FUNCTION_BLOCK fbInverterPosCtrl
VAR_INPUT
	bHomingRdy		:	BOOL;
	bPosStart		:	BOOL;
	dTargetPosNum	:	DINT;
	i1stRPMfix		:	INT;
	i2ndRPMfix		:	INT;
	i2ndSpdRangefix	:	INT;
	iOffSetRangeFix	:	INT;
	iRatioFix			:	REAL;
	lrActualPosition	:	LREAL;

	iPos1			:	INT;
	iPos2			:	INT;
	iPos3			:	INT;
	iPos4			:	INT;
	iPos5			:	INT;
	iPos6			:	INT;
	iPos7			:	INT;
	iPos8			:	INT;
	iPos9			:	INT;
	iPos10			:	INT;
	iPos11			:	INT;
	iPos12			:	INT;
	iPos13			:	INT;
	iPos14			:	INT;
	iPos15			:	INT;
	iPos16			:	INT;
	iPos17			:	INT;
	iPos18			:	INT;
	iPos19			:	INT;
	iPos20			:	INT;


END_VAR
VAR_OUTPUT
	bMoveDone		:	BOOL;
	bMoveFor		: 	BOOL;
	bMoveRev		:	BOOL;
	iTargetPos		:	INT ;

END_VAR
VAR_IN_OUT
	iSpdOut			:	INT;
	PosSv			:	INT;

END_VAR
VAR

	Move_1: AM_MoveAbsolute;
	Move1: BOOL;
	Move2: BOOL;
	Move3: BOOL;
	Move4: BOOL;
	Move5: BOOL;
	Move6: BOOL;
	Move7: BOOL;
	Move8: BOOL;
	Move9: BOOL;
	Move10: BOOL;
	Move11: BOOL;
	Move12: BOOL;
	Move13: BOOL;
	Move14: BOOL;
	Move15: BOOL;
	Move16: BOOL;
	Move17: BOOL;
	Move18: BOOL;
	Move19: BOOL;
	Move20: BOOL;


	ArmMoveStart: BOOL;
	iSpdOutTemp: INT;
	FB: fbArmMoveInterLock;

	ArmMoveEn: BOOL;
	TON1: TON;
	bSpeedNormalEn: BOOL;
	iSlowSpeedRange: INT;

	iDccTime		:	INT := 5;
	iDccStep			:	INT := 2;
END_VAR
VAR // added by the converter: edge detectors and wires of the graphical bodies
    _w1, _w3, _w4, _w5, _w6, _w7, _w8, _w9, _w10, _w11, _w12, _w13, _w14, _w15, _w16, _w17, _w18, _w19, _w20, _w21, _w22 : INT;
    _w2 : ANY;
END_VAR

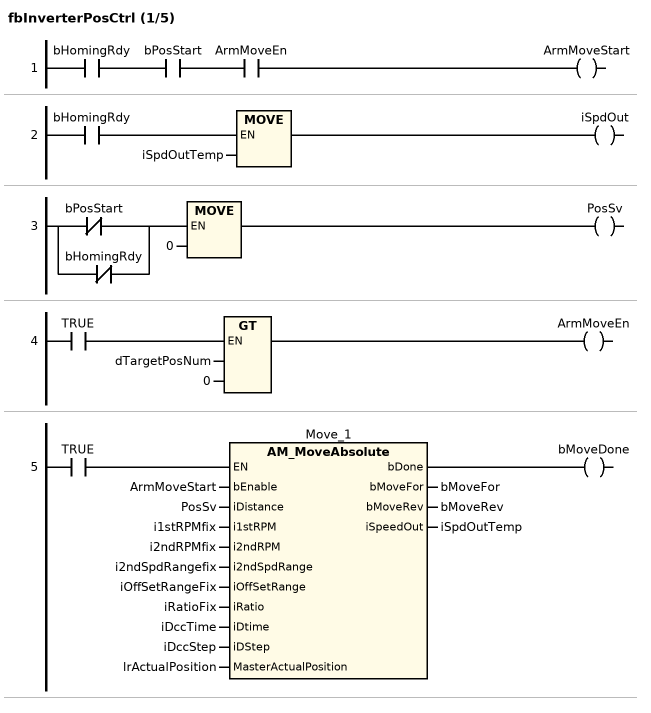
// NETWORK 1
ArmMoveStart := bHomingRdy AND bPosStart AND ArmMoveEn;

// NETWORK 2
IF bHomingRdy THEN _w1 := iSpdOutTemp; END_IF
iSpdOut := _w1;

// NETWORK 3
IF NOT bPosStart OR NOT bHomingRdy THEN _w2 := 0; END_IF
PosSv := _w2;

// NETWORK 4
ArmMoveEn := dTargetPosNum > 0;

// NETWORK 5
Move_1(
    bEnable := ArmMoveStart,
    iDistance := PosSv,
    i1stRPM := i1stRPMfix,
    i2ndRPM := i2ndRPMfix,
    i2ndSpdRange := i2ndSpdRangefix,
    iOffSetRange := iOffSetRangeFix,
    iRatio := iRatioFix,
    iDtime := iDccTime,
    iDStep := iDccStep,
    MasterActualPosition := lrActualPosition,
    bMoveFor => bMoveFor,
    bMoveRev => bMoveRev,
    iSpeedOut => iSpdOutTemp); // AM_MoveAbsolute
bMoveDone := Move_1.bDone;

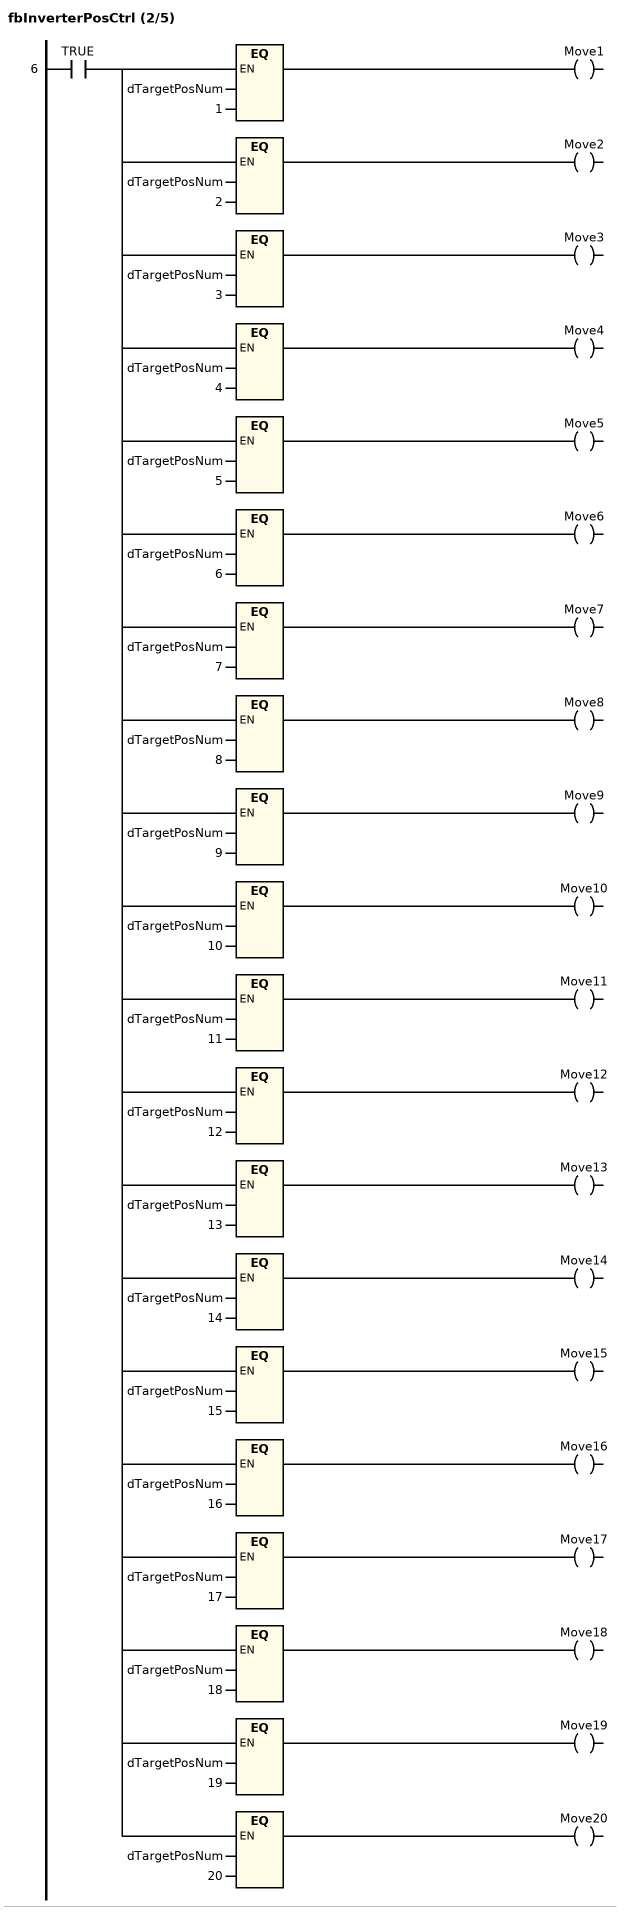
// NETWORK 6
Move1 := dTargetPosNum = 1;
Move2 := dTargetPosNum = 2;
Move3 := dTargetPosNum = 3;
Move4 := dTargetPosNum = 4;
Move5 := dTargetPosNum = 5;
Move6 := dTargetPosNum = 6;
Move7 := dTargetPosNum = 7;
Move8 := dTargetPosNum = 8;
Move9 := dTargetPosNum = 9;
Move10 := dTargetPosNum = 10;
Move11 := dTargetPosNum = 11;
Move12 := dTargetPosNum = 12;
Move13 := dTargetPosNum = 13;
Move14 := dTargetPosNum = 14;
Move15 := dTargetPosNum = 15;
Move16 := dTargetPosNum = 16;
Move17 := dTargetPosNum = 17;
Move18 := dTargetPosNum = 18;
Move19 := dTargetPosNum = 19;
Move20 := dTargetPosNum = 20;

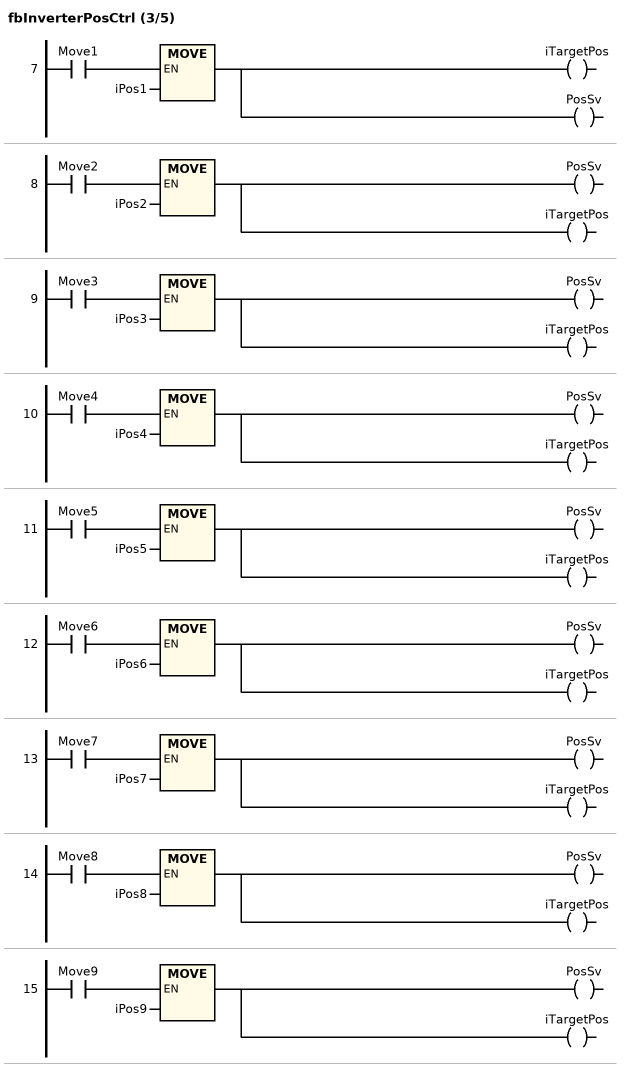
// NETWORK 7
IF Move1 THEN _w3 := iPos1; END_IF
iTargetPos := _w3;
PosSv := _w3;

// NETWORK 8
IF Move2 THEN _w4 := iPos2; END_IF
PosSv := _w4;
iTargetPos := _w4;

// NETWORK 9
IF Move3 THEN _w5 := iPos3; END_IF
PosSv := _w5;
iTargetPos := _w5;

// NETWORK 10
IF Move4 THEN _w6 := iPos4; END_IF
PosSv := _w6;
iTargetPos := _w6;

// NETWORK 11
IF Move5 THEN _w7 := iPos5; END_IF
PosSv := _w7;
iTargetPos := _w7;

// NETWORK 12
IF Move6 THEN _w8 := iPos6; END_IF
PosSv := _w8;
iTargetPos := _w8;

// NETWORK 13
IF Move7 THEN _w9 := iPos7; END_IF
PosSv := _w9;
iTargetPos := _w9;

// NETWORK 14
IF Move8 THEN _w10 := iPos8; END_IF
PosSv := _w10;
iTargetPos := _w10;

// NETWORK 15
IF Move9 THEN _w11 := iPos9; END_IF
PosSv := _w11;
iTargetPos := _w11;

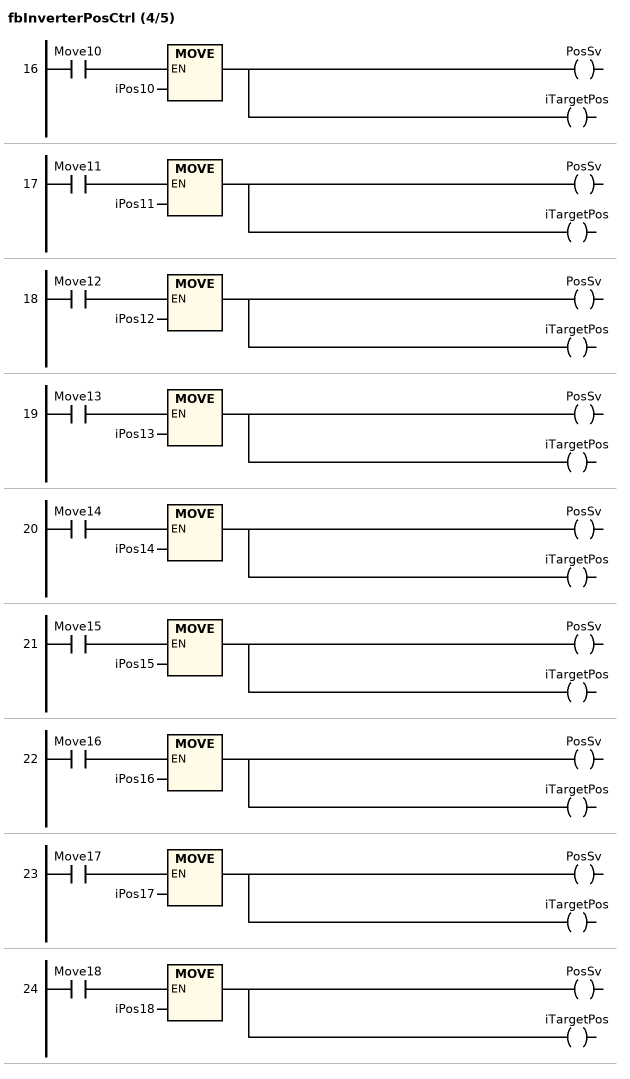
// NETWORK 16
IF Move10 THEN _w12 := iPos10; END_IF
PosSv := _w12;
iTargetPos := _w12;

// NETWORK 17
IF Move11 THEN _w13 := iPos11; END_IF
PosSv := _w13;
iTargetPos := _w13;

// NETWORK 18
IF Move12 THEN _w14 := iPos12; END_IF
PosSv := _w14;
iTargetPos := _w14;

// NETWORK 19
IF Move13 THEN _w15 := iPos13; END_IF
PosSv := _w15;
iTargetPos := _w15;

// NETWORK 20
IF Move14 THEN _w16 := iPos14; END_IF
PosSv := _w16;
iTargetPos := _w16;

// NETWORK 21
IF Move15 THEN _w17 := iPos15; END_IF
PosSv := _w17;
iTargetPos := _w17;

// NETWORK 22
IF Move16 THEN _w18 := iPos16; END_IF
PosSv := _w18;
iTargetPos := _w18;

// NETWORK 23
IF Move17 THEN _w19 := iPos17; END_IF
PosSv := _w19;
iTargetPos := _w19;

// NETWORK 24
IF Move18 THEN _w20 := iPos18; END_IF
PosSv := _w20;
iTargetPos := _w20;

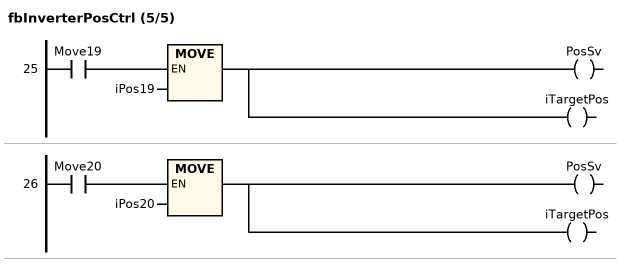
// NETWORK 25
IF Move19 THEN _w21 := iPos19; END_IF
PosSv := _w21;
iTargetPos := _w21;

// NETWORK 26
IF Move20 THEN _w22 := iPos20; END_IF
PosSv := _w22;
iTargetPos := _w22;

END_FUNCTION_BLOCK

(* stored: Version 1.1.0.1, ProductVersion 3.1.4024.12
   POU fbInverterPosCtrl: Id {8b404e8f-9b37-4b83-ba1f-d86240141e0d}, SpecialFunc None *)
